// instrumetn kinematic paramters
TYPE ST_InstruKinematicParam :
STRUCT	
	
	// instrument geometric parameters
	// NOTE: need update based on instrument types
	m_rodLength:LREAL:=0.5392;
	m_headLength:LREAL :=0.01;
	m_fingerLenght:LREAL :=0;
	m_maxGripAngle :LREAL := 60.0 * g_deg2Rad;
	m_minGripAngle :LREAL := -5 * g_deg2Rad; // make sure fingers are fully closed
	
	// instrument kinematic parameters for joint/DH space transformation
	kx:lreal:=1;
	ky:lreal:=1;
	kz:LREAL:=1;
	k13:LREAL:=0.775;
	k23:LREAL:=0.775;
	m_openAngleDir:INT:=-1;

	Len_fixed_point:LREAL:=0.2;	//不动点距离安装面的长度
	Len_mounting_surface:LREAL:=0.009; //器械安装面距离滑块的长度(图中的L3)
	Len_Hight:lreal:=0; //器械杆的高度
	slope_angle:LREAL:=0; //如果器械是摄像头，还需要考虑摄像头的斜面角度
	open_angle_max:LREAL:=1.57;

END_STRUCT
END_TYPE

(* stored: Version 1.1.0.1, ProductVersion 3.1.4024.11
   DUT ST_InstruKinematicParam: Id {c902676e-88fd-4523-9f32-42df361ddc7d} *)
